KUKA KRL data list: A03_grp_global.dat

&ACCESS RVE
&REL 11
&COMMENT V_1_4_0
&PARAM DISKPATH = BMW_App
DEFDAT  A03_GRP_GLOBAL PUBLIC
;********************************
;Date: 07.11.2018
;Programmer: AIUT
;Description: Global positions
;********************************





ENDDAT
